/// machine data that is used through most sequences of the unit (motor speed, axes positions, ...)
TYPE ScriblyDataMachine :
STRUCT
  Slowspeed : LREAL;
  Highspeed : LREAL;
END_STRUCT
END_TYPE

(* stored: Version 1.1.0.1
   DUT ScriblyDataMachine: Id {90b292de-d882-4839-be3b-b44a39ae45a0} *)
